PROGRAM RunGrindingWheel
VAR
END_VAR

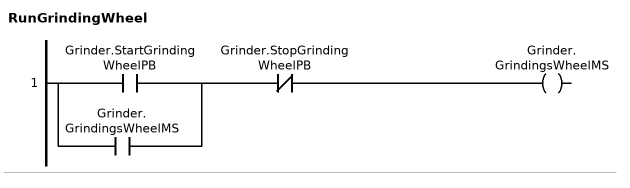
// NETWORK 1
Grinder.GrindingsWheelMS := (Grinder.StartGrindingWheelPB OR Grinder.GrindingsWheelMS) AND NOT Grinder.StopGrindingWheelPB;

END_PROGRAM

(* stored: Version 1.1.0.1, ProductVersion 3.1.4020.12
   POU RunGrindingWheel: Id {d2fda1fb-7af8-4599-b8be-4a9cab5cdfc0}, SpecialFunc None *)
